{attribute addProperty BoxType "AT2040-0250-0022"}
{attribute addProperty Id "A_0107_AT2000_5233_0018_AT2000_5233AT2000_3DCFC8D064080"}
{attribute addProperty CRC "4114873715"}
{attribute addProperty SizeInBites "640"}
{attribute addProperty SizeInBytes "80"}
TYPE A_0037_AT2040_0250_0022_F543FD73 EXTENDS AT2040_9506A482 :
STRUCT
	{attribute addProperty Name "A_0107_AT2000_5233_0018_AT2000_5233"}
	A_0107_AT2000_5233_0018_AT2000_5233 : AT2000_3DCFC8D0;
END_STRUCT
END_TYPE

(* stored: Version 1.2.0.0, ProductVersion 3.1.4024.9
   DUT A_0037_AT2040_0250_0022_F543FD73: Id {8c3428e5-de7f-4d15-8b20-cc5595feff1d} *)
